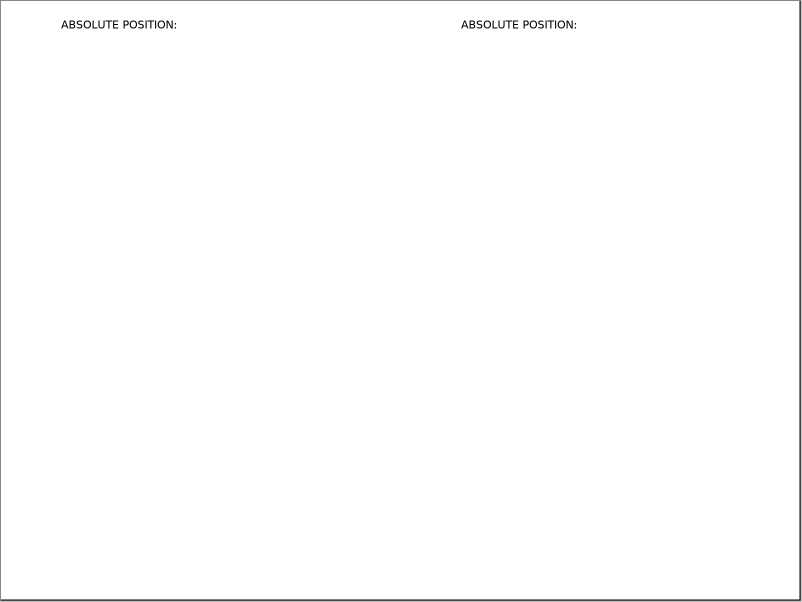
VISUALIZATION F43_Gear_Out  // 802x602
    Rectangle (0,0 800x600)
    Label (10,10 170x30), "ABSOLUTE POSITION:"
    Label (410,10 170x30), "ABSOLUTE POSITION:"
END_VISUALIZATION

(* stored: Version 1.1.0.1, ProductVersion 3.1.4022.7
   Visu F43_Gear_Out: Id {e66ca285-af50-480d-a7d8-b2c466757d1d} *)
